TYPE AxesRotationAxisStatuses :
STRUCT
	///Is the axis in a busy state?
	busyStatus: BusyStatus;
	///Is the axis in a healthy state?
	healthStatus: HealthStatus;
	///Is the axis powered on or off?
	poweredStatus: PoweredStatus;
END_STRUCT
END_TYPE

(* stored: Version 1.1.0.1, ProductVersion 3.1.4019.2
   DUT AxesRotationAxisStatuses: Id {79695c7e-d51b-454b-bc95-d912891803e6} *)
